(* IEC 61131-3 sources: CodesysTest/alpha/export/FBs/Fault/FB_Fault.pou, 5 files *)

(* ---- FB_Fault.pou.st ---- *)
(*#-#-#-#-#-#-#-#-#-#---Declaration---#-#-#-#-#-#-#-#-#-#-#-#-#*)

FUNCTION_BLOCK FINAL FB_Fault IMPLEMENTS IFault, ILoggable, IExecuteAutomatically
VAR_INPUT
	faultTrigger : BOOL;

END_VAR
VAR_OUTPUT
	active : BOOL;
END_VAR
VAR
	_ack : BOOL;
	_acked : BOOL;
	_passive : BOOL;
	_exitConveyorOverride : BOOL;
	_externalExitConveyorOverride : BOOL;
	_logger : IMachineLogger;
	_ackOSR : Standard.R_TRIG;
	_activeONS : FB_ONS;
	_faultTriggerONS : FB_ONS;
	_passiveOSF : Standard.F_TRIG;
	_passiveTimeout : Standard.TON;
	_timeoutDwell : REAL;
	_triggerRequiredToMoveToActiveFaults : PASSIVE_FAULT_TRIGGERS;
	_instanceName : STRING;
	_isOEEExempt : BOOL;
	_isPassiveExempt : BOOL;
END_VAR(*#-#-#-#-#-#-#-#-#-#---Implementation---#-#-#-#-#-#-#-#-#-#-#-#-#*)

(* ---- Ack.m.st ---- *)
(*#-#-#-#-#-#-#-#-#-#---Declaration---#-#-#-#-#-#-#-#-#-#-#-#-#*)

METHOD Ack(*#-#-#-#-#-#-#-#-#-#---Implementation---#-#-#-#-#-#-#-#-#-#-#-#-#*)

IF _ack OR _acked THEN
	RETURN;
END_IF
_acked := TRUE;
// Log the ACK.
_logger.AddLogItem(CONCAT(InstanceName,  ' Acked'));

(* ---- Execute.m.st ---- *)
(*#-#-#-#-#-#-#-#-#-#---Declaration---#-#-#-#-#-#-#-#-#-#-#-#-#*)

METHOD Execute
(*#-#-#-#-#-#-#-#-#-#---Implementation---#-#-#-#-#-#-#-#-#-#-#-#-#*)

//	Function Block: FB_Fault
//	Description: Faults should be of this FB type.
//	Implementation should look as follows:
//
//  *** Instantiate the fault with constructor that contains the fault name: ***
//  VAR (*Faults*)
//		exampleFault1 : FB_Fault(name := CONCAT(_prefix,  'Example Fault 1'));
//		exampleFault2 : FB_Fault(name := CONCAT(_prefix,  'Example Fault 2'));
//  END_VAR
//
//	*** Either assign faultTrigger in call or set it later in logic
//	exampleFault1.faultTrigger := someFaultCondition;
//
//	Created by: Ben Hess
//	Created Date: Tuesday, May 22, 2018

//
_passiveOSF(CLK := _passive);

//
_passiveTimeout(IN := _passive, PT := TO_TIME(_timeoutDwell * 1000));
IF _passiveTimeout.Q THEN
	THIS^.Trigger();
	_passive := FALSE;
END_IF

//
_faultTriggerONS(CLK := faultTrigger);
IF _faultTriggerONS.OSR THEN
	Trigger();
END_IF

//
_ackOSR(CLK := _ack);
IF _ackOSR.Q THEN
	_acked := TRUE;
	_ack := FALSE;
END_IF

//
IF _acked THEN
	_acked := FALSE;
	IF NOT faultTrigger THEN
		active := FALSE;
	END_IF
	_passive := FALSE;
END_IF

//
_activeONS(CLK := active);
IF _activeONS.OSF THEN
	GlobalObjects.CollectionOfActiveFaults.RemoveObject(THIS^);
	IF _isOEEExempt THEN
		GlobalObjects.CollectionOfOEEExemptFaults.RemoveObject(THIS^);
	END_IF
	IF _isPassiveExempt THEN
		GlobalObjects.CollectionOfPassiveExemptFaults.RemoveObject(THIS^);
	END_IF
	_logger.AddLogItem(CONCAT(InstanceName, ' Active Cleared'));
ELSIF _activeONS.OSR OR _passiveOSF.Q THEN
	GlobalObjects.CollectionOfPassiveFaults.RemoveObject(THIS^);
	//_logger.AddLogItem(CONCAT(InstanceName, ' Passive Cleared'));
END_IF

(* ---- FB_Init.m.st ---- *)
(*#-#-#-#-#-#-#-#-#-#---Declaration---#-#-#-#-#-#-#-#-#-#-#-#-#*)

METHOD FB_Init : BOOL
VAR_INPUT
  bInitRetains : BOOL; // TRUE: the retain variables are initialized (reset warm / reset cold)
  bInCopyCode : BOOL;  // TRUE: the instance will be copied to the copy code afterward (online change)
  name : STRING;
END_VAR
VAR
	_j : DINT;
	_totalOEEExempt : DINT := GlobalObjects.OEE_EXEMPT_LIST_LENGTH;
	_totalPassiveExempt : DINT := GlobalObjects.PASSIVE_EXEMPT_LIST_LENGTH;
END_VAR
(*#-#-#-#-#-#-#-#-#-#---Implementation---#-#-#-#-#-#-#-#-#-#-#-#-#*)

_instanceName := name;
GlobalObjects.CollectionOfAllObjects.AddObject(THIS^);
FOR _j := 1 TO _totalOEEExempt DO
	IF GlobalObjects.OEEExemptList[_j] = name THEN
		_isOEEExempt := TRUE;
	END_IF
END_FOR

FOR _j := 1 TO _totalPassiveExempt DO
	IF GlobalObjects.passiveList[_j] = name THEN
		_isPassiveExempt := TRUE;
	END_IF
END_FOR

(* ---- Trigger.m.st ---- *)
(*#-#-#-#-#-#-#-#-#-#---Declaration---#-#-#-#-#-#-#-#-#-#-#-#-#*)

METHOD Trigger
(*#-#-#-#-#-#-#-#-#-#---Implementation---#-#-#-#-#-#-#-#-#-#-#-#-#*)

IF active = TRUE THEN
	RETURN;
END_IF
active := TRUE;
GlobalObjects.CollectionOfActiveFaults.AddObject(THIS^);
IF _isOEEExempt THEN
	GlobalObjects.CollectionOfOEEExemptFaults.AddObject(THIS^);
END_IF
IF _isPassiveExempt THEN
	GlobalObjects.CollectionOfPassiveExemptFaults.AddObject(THIS^);
END_IF
IF _logger <> 0 THEN
	_logger.AddLogItem(CONCAT(InstanceName,  ' Active'));
END_IF
